// TwinCAT 3 PLC project CNCControl
// ProgramVersion: 3.1.4022.4
// libraries:
//   Tc2_EthernetIP, * (Beckhoff Automation GmbH)
//   Tc2_IoFunctions, * (Beckhoff Automation GmbH)
//   Tc2_Math, * (Beckhoff Automation GmbH)
//   Tc2_Standard, * (Beckhoff Automation GmbH)
//   Tc2_System, * (Beckhoff Automation GmbH)
//   Tc2_Utilities, * (Beckhoff Automation GmbH)
//   Tc3_Module, * (Beckhoff Automation GmbH)
// project tree:
//   DUTs/ E_CIA402State.TcDUT (not stored), E_PIDOptimizationStage.TcDUT (not stored), E_PIDOptimizationType.TcDUT
//   / EveryHundredMilliseconds.TcTTO, EveryMS.TcTTO, MainCNCControl.TcTTO
//   GVLs/ Constants.TcGVL
//   POUs/ MAIN.TcPOU
//   POUs/SpindleSpeed/ AnalogDemandedSpeedCalculator.TcPOU, AnalogPrescaledSpeedCalculator.TcPOU, DemandedSpeedInterface.TcIO, DemandedSpeedTask.TcPOU, PWMDemandedSpeedCalculator.TcPOU, SpindleSpeedCalculator.TcPOU
//   POUs/Spindle/ SpindleCIA402Velocity.TcPOU, SpindleController.TcIO, SpindleDeltaVFDOverEIP.TcPOU
//   POUs/Utilities/ FB_FreqMeasure.TcPOU, FB_MovingAverageUInt.TcPOU, FB_MovingAverageReal.TcPOU, FB_OptimizePID.TcPOU, FB_ScaleBetween.TcPOU
//   POUs/Vacuum/ VacuumATV71Ethercat.TcPOU, FB_GetVacuumAMSID.TcPOU (not stored), ToshibaP9VacuumPressureGetter.TcPOU (not stored), VacuumController.TcIO
// real-time tasks:
//   TASK EveryHundredMilliseconds: cycle T#100000us, priority 10, ADS port 350
//   TASK MainCNCControl: cycle T#1ms, priority 6, ADS port 351
//   TASK EveryMS: cycle T#1ms, priority 4, ADS port 352
// I/O:
//   DEVICE Device 1 (EtherCAT), AmsNetId 192.168.1.51.2.1
//     Box 16 (ATV71 EtherCAT) [ATV71 EtherCAT]
//     HITECO UE-1F 6.6 Spindle [KEB_F6_drive_unit_EtherCAT]
//     Term 1 (EK1100) [EK1100 EtherCAT Coupler (2A E-Bus)]
//       Term 3 (EL1502) [EL1502 2Ch. +/- Counter 24V, 100kHz]
//       Term 4 (EL1809) [EL1809 16Ch. Dig. Input 24V, 3ms]
//       Term 5 (EL1889) [EL1889 16Ch. Dig. Input 24V, 3ms, negative]
//       Term 15 (EL1018) [EL1018 8Ch. Dig. Input 24V, 10µs]
//       Term 20 (EL9110) [EL9110 Power Supplier with LED (24V, Diagnostics)]
//       Term 19 (EL2622) [EL2622 2Ch. Relay Output, NO (230V AC / 30V DC)]
//       Term 26 (EL6070) [EL6070 1Ch. Licensing-Terminal]
//       Term 6 (EL9400) [EL9400 E-Bus Power Supplier]
//       Term 27 (EL1262-0050) [EL1262-0050 2Ch. Dig. Input 5V, 1µs, DC Oversample]
//       Term 7 (EL2124) [EL2124 4Ch. Dig. Output 5V, 20mA]
//       Term 8 (EL2124) [EL2124 4Ch. Dig. Output 5V, 20mA]
//       Term 9 (EL2124) [EL2124 4Ch. Dig. Output 5V, 20mA]
//       Term 10 (EL1124) [EL1124 4Ch. Dig. Input 5V, 10µs, Sensor Power]
//       Term 11 (EL1124) [EL1124 4Ch. Dig. Input 5V, 10µs, Sensor Power]
//       Term 12 (EL9011) [EL9011 End Terminal]
//   DEVICE Device 2 (TC3 EIP Scanner), AmsNetId 192.168.1.51.3.1
//     Box 12 (Nitra CMV EtherNet/IP) // <INFO> </INFO> <EDS> C:\TwinCAT\3.1\Config\Io\EtherNetIP\nitraethernetip.eds </EDS>
//     Box 13 (IPE001Z) (disabled) // <INFO> </INFO> <EDS> C:\TwinCAT\3.1\Config\Io\EtherNetIP\IPE001Z_AS1.eds </EDS>
//     Box 2 (CMM-EIP01) (disabled) // <INFO> </INFO> <EDS> C:\TwinCAT\3.1\Config\Io\EtherNetIP\031F000C010400010001.eds </EDS>
// variable links:
//   CNCControl/CNCControl Instance <-> Device 1 (EtherCAT)/Box 16 (ATV71 EtherCAT)
//     MainCNCControl Inputs/MAIN.VacuumControl.iAnalogInput2ScaledValue <-> Inputs/MAIN.VacuumControl.iAnalogInput2ScaledValue
//     MainCNCControl Inputs/MAIN.VacuumControl.iOutputFrequency <-> Inputs/MAIN.VacuumControl.iOutputFrequency
//     MainCNCControl Inputs/MAIN.VacuumControl.iOutputVelocity <-> Inputs/MAIN.VacuumControl.iOutputVelocity
//     MainCNCControl Inputs/MAIN.VacuumControl.iPIDRegulatorFeedback <-> Inputs/MAIN.VacuumControl.iPIDRegulatorFeedback
//     MainCNCControl Inputs/MAIN.VacuumControl.iPIDRegulatorOutput <-> Inputs/MAIN.VacuumControl.iPIDRegulatorOutput
//     MainCNCControl Inputs/MAIN.VacuumControl.iStatusWord <-> Inputs/MAIN.VacuumControl.iStatusWord
//     MainCNCControl Outputs/MAIN.VacuumControl.oMotorFrequency <-> Outputs/MAIN.VacuumControl.oMotorFrequency
//     MainCNCControl Outputs/MAIN.VacuumControl.oVacuumControl <-> Outputs/MAIN.VacuumControl.oVacuumControl
//     MainCNCControl Outputs/MAIN.VacuumControl.oVacuumPressureRequested <-> Outputs/MAIN.VacuumControl.oVacuumPressureRequested
//   CNCControl/CNCControl Instance <-> Device 1 (EtherCAT)/HITECO UE-1F 6.6 Spindle
//     MainCNCControl Inputs/MAIN.SpindleControl.iStatusWord <-> Inputs/statusword [0x6041.0]
//     MainCNCControl Outputs/MAIN.SpindleControl.oControlWord <-> Outputs/controlword [0x6040.0]
//     MainCNCControl Outputs/MAIN.SpindleControl.oTargetVelocity <-> Outputs/vl target velocity [0x6042.0]
//   CNCControl/CNCControl Instance <-> Device 1 (EtherCAT)/Term 1 (EK1100)/Term 11 (EL1124)
//     MainCNCControl Inputs/MAIN.iPCCoolantOn <-> Channel 4/MAIN.iPCCoolantOn
//     MainCNCControl Inputs/MAIN.iPCSpindleOn <-> Channel 1/MAIN.iPCSpindleOn
//     MainCNCControl Inputs/MAIN.iPCToolRelease <-> Channel 3/MAIN.iPCToolRelease
//     MainCNCControl Inputs/MAIN.iPCVacuumOn <-> Channel 2/MAIN.iPCVacuumOn
//   CNCControl/CNCControl Instance <-> Device 1 (EtherCAT)/Term 1 (EK1100)/Term 15 (EL1018)
//     MainCNCControl Inputs/MAIN.iProbe <-> Channel 1/MAIN.iProbe
//   CNCControl/CNCControl Instance <-> Device 1 (EtherCAT)/Term 1 (EK1100)/Term 19 (EL2622)
//     MainCNCControl Outputs/MAIN.oZAxisBrakeRelay <-> Channel 1/MAIN.oZAxisBrakeRelay
//   CNCControl/CNCControl Instance <-> Device 1 (EtherCAT)/Term 1 (EK1100)/Term 27 (EL1262-0050)
//     EveryMS Inputs/DemandedSpeedTask.DemandedSpeedImpl.iInputSpeedBits[{1..125}] <-> Ch1 Input {0..124}/Ch1 Input  (125 links)
//   CNCControl/CNCControl Instance <-> Device 1 (EtherCAT)/Term 1 (EK1100)/Term 3 (EL1502)
//     EveryHundredMilliseconds Inputs/SpindleSpeedCalculator.CounterValue <-> CNT Inputs Channel 1/Counter value
//   CNCControl/CNCControl Instance <-> Device 1 (EtherCAT)/Term 1 (EK1100)/Term 4 (EL1809)
//     MainCNCControl Inputs/MAIN.iAirPressureSensor <-> Channel 1/MAIN.iPressureSensor
//     MainCNCControl Inputs/MAIN.iS1ToolPresence <-> Channel 5/MAIN.iS1ToolPresence
//     MainCNCControl Inputs/MAIN.iS2ColletOpen <-> Channel 4/MAIN.iS2ColletOpen
//     MainCNCControl Inputs/MAIN.iSpindleOverTemp <-> Channel 3/MAIN.iSpindleOverTemp
//     MainCNCControl Inputs/MAIN.iSpindleToolReleaseButton <-> Channel 2/MAIN.iSpindleToolReleaseButton
//   CNCControl/CNCControl Instance <-> Device 1 (EtherCAT)/Term 1 (EK1100)/Term 5 (EL1889)
//     MainCNCControl Inputs/MAIN.iAAxisAlarm <-> Channel 5/Input
//     MainCNCControl Inputs/MAIN.iXAxisAlarm <-> Channel 2/MAIN.iXAxisAlarm
//     MainCNCControl Inputs/MAIN.iYAxisAlarm <-> Channel 1/MAIN.iYAxisAlarm
//     MainCNCControl Inputs/MAIN.iZAxisAlarm <-> Channel 3/MAIN.iZAxisAlarm
//     MainCNCControl Inputs/MAIN.iZAxisBrakeOff <-> Channel 4/MAIN.iZAxisBrakeOff
//   CNCControl/CNCControl Instance <-> Device 1 (EtherCAT)/Term 1 (EK1100)/Term 7 (EL2124)
//     MainCNCControl Outputs/MAIN.oPCToolPresence <-> Channel 4/MAIN.PCToolPresence
//   CNCControl/CNCControl Instance <-> Device 1 (EtherCAT)/Term 1 (EK1100)/Term 8 (EL2124)
//     MainCNCControl Outputs/MAIN.oPCColletOpen <-> Channel 2/MAIN.oPCColletOpen
//     MainCNCControl Outputs/MAIN.oPCServoAlarm <-> Channel 1/MAIN.oPCServoAlarm
//     MainCNCControl Outputs/MAIN.oPCSpindleStopped <-> Channel 3/MAIN.oPCSpindleStopped
//     MainCNCControl Outputs/MAIN.oPCVacuumPressureGood <-> Channel 4/MAIN.oPCVacuumPressureGood
//   CNCControl/CNCControl Instance <-> Device 1 (EtherCAT)/Term 1 (EK1100)/Term 9 (EL2124)
//     MainCNCControl Outputs/MAIN.oPCAirPressure <-> Channel 1/MAIN.oPCAirPressure
//     MainCNCControl Outputs/MAIN.oPCProbe <-> Channel 2/MAIN.oPCProbe
//     MainCNCControl Outputs/MAIN.oPCSpindleOverTemp <-> Channel 4/MAIN.oPCSpindleOverTemp
//     MainCNCControl Outputs/MAIN.oPCSpindleSpeedOK <-> Channel 3/MAIN.oPCSpindleSpeedOK
//   CNCControl/CNCControl Instance <-> Device 2 (TC3 EIP Scanner)/Box 12 (Nitra CMV EtherNet/IP)
//     MainCNCControl Outputs/MAIN.oValveControl <-> Connection 1 (Input/Output)/Outputs/MAIN.oValveControl

CONFIGURATION CNCControl
    RESOURCE PLC ON TwinCAT3
        TASK EveryHundredMilliseconds(INTERVAL := T#100000us, PRIORITY := 10);
        TASK EveryMS(INTERVAL := T#1ms, PRIORITY := 4);
        TASK MainCNCControl(INTERVAL := T#1ms, PRIORITY := 6);
        PROGRAM VacuumPressureGetter WITH EveryHundredMilliseconds : VacuumPressureGetter;
        PROGRAM SpindleSpeedCalculator WITH EveryHundredMilliseconds : SpindleSpeedCalculator;
        PROGRAM DemandedSpeedTask WITH EveryMS : DemandedSpeedTask;
        PROGRAM MAIN WITH MainCNCControl : MAIN;
    END_RESOURCE
END_CONFIGURATION

// ---- DUTs/E_PIDOptimizationType.TcDUT
{attribute 'qualified_only'}
{attribute 'strict'}
TYPE E_PIDOptimizationType :
(
	NoOvershoot,
	SomeOvershoot,
	FastRamp
);
END_TYPE

// ---- GVLs/Constants.TcGVL
{attribute 'qualified_only'}
VAR_GLOBAL CONSTANT
	// Number of RPM per HZ in the VFD
	RPMPerHZ : UINT := 30;
	// VFD frequency precision in 1/X of 1 HZ. So 10 means it can do 1/10th of a HZ
	VFDHZPrecision : UINT := 10;
	// Minimum VFD RPM increment based on RPM per HZ and precision
	VFDMinRPMIncrement : UINT := TO_UINT(RPMPerHZ / VFDHZPrecision);
	// One second in microseconds
	OneSecondInUs : UDINT := 1000000;
END_VAR

// ---- POUs/SpindleSpeed/DemandedSpeedInterface.TcIO
INTERFACE DemandedSpeedInterface

METHOD GetSpeed : UINT
END_METHOD

END_INTERFACE

// ---- POUs/Spindle/SpindleController.TcIO
INTERFACE SpindleController

METHOD Run : BOOL
END_METHOD

METHOD SetDirection : BOOL
VAR_INPUT
	// Set the spindle rotation direction
	Reverse : BOOL;
END_VAR
END_METHOD

METHOD SetSpeed : BOOL
VAR_INPUT
	Speed : UINT;
END_VAR
END_METHOD

METHOD Stop : BOOL
END_METHOD

END_INTERFACE

// ---- POUs/Vacuum/VacuumController.TcIO
INTERFACE VacuumController

METHOD GetCurrentPressure : REAL
END_METHOD

METHOD Run : BOOL
END_METHOD

METHOD SetPressureRequired : BOOL
VAR_INPUT
	Pressure : REAL;
END_VAR
END_METHOD

METHOD Stop : BOOL
END_METHOD

END_INTERFACE

// ---- POUs/SpindleSpeed/SpindleSpeedCalculator.TcPOU
PROGRAM SpindleSpeedCalculator
VAR
	// Spindle speed in RPM
	{attribute 'UserUnit' := '<AngularVelocity, RPM, RPM, 9.549296596425, 0, 0 >'}
	SpindleSpeed : LREAL;
	// Current pulse count value from the counter
	PulseCount: UINT;
	// Counter value from previous time we read the counter
	LastCounterValue: UDINT;
	// Counter value from counter
	CounterValue AT %I*: UDINT;
	// Array of spindle speeds
	SpindleSpeeds : ARRAY[0..4] OF LREAL;
	MovingAverage : FB_MovingAverageReal;
END_VAR
VAR_TEMP
	TempSpindleSpeed: REAL;
END_VAR
VAR CONSTANT
	// Pulses per revolution of the spindle sensor
	PulsesPerRevolution : UINT := 2;
	// Task cycles per minute - task runs every 100ms
	TaskCyclesPerMinute : UINT := 600;
END_VAR

// Convert counter value to pulses since last cycle
PulseCount := TO_UINT(CounterValue - LastCounterValue);
LastCounterValue := CounterValue;
// Extrapolate how pulses many would have occurred in a minute, then divide by pulses per revolution to get RPM.
TempSpindleSpeed := (TO_REAL(PulseCount) * TaskCyclesPerMinute) / PulsesPerRevolution;
MovingAverage(ValueToAdd := TempSpindleSpeed,
			  AverageArray := SpindleSpeeds);
SpindleSpeed := MovingAverage.CurrentValue;

END_PROGRAM

// ---- POUs/Utilities/FB_MovingAverageReal.TcPOU
FUNCTION_BLOCK FB_MovingAverageReal
VAR_INPUT
	ValueToAdd : LREAL;
END_VAR
VAR_IN_OUT
	AverageArray  : ARRAY [*] OF LREAL;
END_VAR
VAR_OUTPUT
	CurrentValue : LREAL;
END_VAR
VAR
	CurrentIndex : UINT;
	NumValues: UINT;
END_VAR
VAR_TEMP
	Counted : UINT;
	I: DINT;
	Sum: LREAL;
	ArrayLength : UINT;
END_VAR

// Compute average over array.
// The order of this addition and MOD are important to avoid going out of bounds.
// NOTE: We deliberately do not try to account for underfilling the array.
ArrayLength := TO_UINT(UPPER_BOUND(AverageArray, 1) - LOWER_BOUND(AverageArray, 1) + 1);
AverageArray[CurrentIndex] := ValueToAdd;
CurrentIndex := CurrentIndex + 1;
CurrentIndex := CurrentIndex MOD ArrayLength;
NumValues := MIN(NumValues + 1 , ArrayLength);
IF NumValues > 0 THEN
	FOR I := LOWER_BOUND(AverageArray, 1) TO UPPER_BOUND(AverageArray, 1) BY 1 DO
		Sum := Sum + AverageArray[I];
		Counted := Counted + 1;
		// Don't count more than the number of values
		IF Counted > NumValues THEN
			EXIT;
		END_IF
	END_FOR
END_IF
CurrentValue := TO_REAL(Sum / NumValues);

END_FUNCTION_BLOCK

// ---- POUs/SpindleSpeed/DemandedSpeedTask.TcPOU
PROGRAM DemandedSpeedTask
VAR
	{attribute 'UserUnit' := '<AngularVelocity, RPM, RPM, 9.549296596425, 0, 0 >'}
	DemandedSpeed : UINT;
	DemandedSpeedImpl : PWMDemandedSpeedCalculator;
END_VAR

DemandedSpeed := DemandedSpeedImpl.GetSpeed();

END_PROGRAM

// ---- POUs/SpindleSpeed/PWMDemandedSpeedCalculator.TcPOU
FUNCTION_BLOCK FINAL PWMDemandedSpeedCalculator IMPLEMENTS DemandedSpeedInterface
VAR
	iInputSpeedBits AT %I* : ARRAY [1..BitArraySize] OF BYTE;
END_VAR
VAR CONSTANT
	// Array Length
	BitArraySize : UINT := 125;
	// PWM frequency
	PWMFrequency : UINT := 200;
    // PWM period
	PWMPeriod : REAL := 1 / PWMFrequency;
	// Microseconds in Frequency
	UsInFrequency : UDINT :=  Constants.OneSecondInUs / PWMFrequency;	
END_VAR

METHOD GetSpeed : UINT
VAR_INST
	TempSpindleSpeed : UINT;
	LastDemandedSpeed : UINT;
	TotalOnTime : UDINT;
	TotalOffTime : UDINT;
	DutyCycle : LREAL;
	DutyCycles : ARRAY [0..20] OF LREAL;
	MovingAverage : FB_MovingAverageReal;
	Scaling : FB_ScaleBetween;
END_VAR
VAR
	I : UINT;	
	J: UINT;
	BitMask : UINT;
	MaskedBit : BOOL;
END_VAR
// The input here is a PWM signal with a frequency of 200, a low of 1% duty, and a high of 95% duty.
// Basic Calculation for PWM pulses

 FOR I := 1 TO BitArraySize BY 1 DO
	 FOR J := 0 TO 7 BY 1 DO
		BitMask := SHL(1, J);
		MaskedBit := TO_BOOL(iInputSpeedBits[I] AND BitMask);
		IF MaskedBit THEN
			TotalOnTime := TotalOnTime + 1;
		ELSE
			TotalOffTime := TotalOffTime + 1; 
		END_IF
		// Stop at the end of the period
		IF (TotalOnTime + TotalOffTime) > UsInFrequency THEN
			EXIT;
		END_IF 
	 END_FOR
 END_FOR
 
// See if the period is up
IF (TotalOnTime + TotalOffTime) > UsInFrequency  THEN
	DutyCycle := TO_LREAL(TotalOnTime) / TO_LREAL(TotalOnTime + TotalOffTime);
	TotalOnTime := 0;
	TotalOffTime := 0;
	// Average the duty cycle and then scale the average
	MovingAverage(ValueToAdd := DutyCycle, 
				  AverageArray := DutyCycles);
	Scaling(RawValue:=MovingAverage.CurrentValue, RawValueMin:=0.0, 
					  RawValueMax:=1, ScaledValueMin:=0,
					  ScaledValueMax:=24000);
	LastDemandedSpeed := TO_UINT(Scaling.ScaledValue);
	// Make sure demanded speed is some increment of what the VFD can do. 
	LastDemandedSpeed := (LastDemandedSpeed / Constants.VFDMinRPMIncrement) * Constants.VFDMinRPMIncrement;
END_IF
GetSpeed := LastDemandedSpeed;
END_METHOD

END_FUNCTION_BLOCK

// ---- POUs/Utilities/FB_ScaleBetween.TcPOU
FUNCTION_BLOCK FB_ScaleBetween
VAR_INPUT
	RawValue : LREAL;
	RawValueMin: LREAL;
	RawValueMax : LREAL;
	ScaledValueMin : LREAL;
	ScaledValueMax : LREAL;
END_VAR
VAR_OUTPUT
	ScaledValue : LREAL;
END_VAR
VAR
END_VAR

ScaledValue :=  (((ScaledValueMax-ScaledValueMin) * (RawValue - RawValueMin)) / (RawValueMax - RawValueMin)) + ScaledValueMin;
ScaledValue := LIMIT(ScaledValueMin, ScaledValue, ScaledValueMax);

END_FUNCTION_BLOCK

// ---- POUs/MAIN.TcPOU
PROGRAM MAIN
VAR
	{region "Servo handling variables"}
	// Alarm inputs from Servos
  	iXAxisAlarm AT %I*:BOOL;
  	iYAxisAlarm AT %I*:BOOL;
  	iZAxisAlarm AT %I*:BOOL;
  	iAAxisAlarm AT %I*:BOOL;
  	// Alarm Output to PC pin 8
  	oPCServoAlarm AT %Q*:BOOL;
  	// Whether servo thinks Z Axis break should be off
  	iZAxisBrakeOff AT %I*:BOOL;
	// Relay output controlling Z Axis Brake
	oZAxisBrakeRelay AT %Q*: BOOL;
    {endregion}
	{region "Probe, Air Pressure, Coolant"}
	// Digital Probe Trigger output to PC pin 29
	oPCProbe AT %Q*: BOOL;
	// Digital Probe Input (Normally Closed)
	iProbe AT %I*: BOOL := TRUE;
	// Air Pressure >90psi signal to PC pin 10
	oPCAirPressure AT %Q*: BOOL;
	// Air Pressure >90psi signal from sensor.  The sensor triggers as pressure is rising past 90psi
	iAirPressureSensor AT %I*: BOOL;
	// Control of NITRA Valves over ethernet/ip	 
	oValveControl AT %Q* : NitraValves; 
	// Turn on coolant signal from PC
	iPCCoolantOn AT %I* : BOOL;
	{endregion}
	{region "Vacuum"}
	VacuumControl: VacuumATV71Ethercat;
	 // Turn on vacuum signal from PC
	iPCVacuumOn AT %I* : BOOL;
	// Vacuum Pressure good output to PC Pin 7
	oPCVacuumPressureGood AT %Q*: BOOL;
	{endregion}
	{endregion}
	{endregion}
	{region "Spindle variables"}
	{region "Spindle Speed Handling"}
	// True if spindle is at less than 1 RPM
	SpindleStopped : BOOL;
	// Spindle stopped output to PC pin 1
	oPCSpindleStopped AT %Q* : BOOL;
	// Spindle within 5% of speed to PC Pin 28
	oPCSpindleSpeedOK AT %Q* : BOOL;
	{endregion}
	{region "Spindle Tool Change handling"}
	// Tool Release Button on Spindle
	iSpindleToolReleaseButton AT %I*: BOOL;
	// Tool Release from PC Pin 24
	iPCToolRelease AT %I*: BOOL;
	// Tool Presence to PC Pin 2
	oPCToolPresence AT %Q* : BOOL;
	// S1 Tool Presence sensor from the spindle
	iS1ToolPresence AT %I* : BOOL;
	// Collet Open to PC Pin 9
	oPCColletOpen AT %Q* : BOOL;
	// S2 Collet Open sensor from the spindle
	iS2ColletOpen AT %I* : BOOL;	 
	// Spindle over temperature to PC Pin 27
	oPCSpindleOverTemp AT %Q* : BOOL;
	// Spindle over temperature relay
	iSpindleOverTemp AT %I* : BOOL;
	// Turn spindle on input from PC
	iPCSpindleOn AT %I* : BOOL;
	SpindleControl : SpindleCIA402Velocity;
	{endregion}
	{endregion}
	{region "Input Debouncers"}
	(* The 5V input has a ridiculously fast time - a few nanoseconds.
	   Therefore, we debounce it *)
	CoolantOnDebounced : TON;
	SpindleOnDebounced : TON;
	ToolReleaseDebounced : TON;	
	VacuumOnDebounced : TON;
	{endregion}
END_VAR
VAR CONSTANT
	// Minimum PSI at which vacuum holding is viable for workpiece
	GoodVacuumPressure : REAL := 10.0;
END_VAR

CoolantOnDebounced(IN := iPCCoolantOn, PT := T#3MS);
SpindleOnDebounced(IN := iPCSpindleOn, PT := T#3MS);
ToolReleaseDebounced(IN := iPCToolRelease, PT := T#3MS);
VacuumOnDebounced(IN := iPCVacuumOn, PT := T#3MS);

{region "Servo handling"}
// Servo Alarm
	// The servo alarm inputs are normally closed
	oPCServoAlarm := NOT (iXAxisAlarm AND_THEN iYAxisAlarm AND_THEN iZAxisAlarm AND_THEN iAAxisAlarm);

// Servo Brake	 
	oZAxisBrakeRelay := iZAxisBrakeOff;
{endregion}

{region "Probe, Air Pressure, Coolant, Vacuum"}
// Probe control
	oPCProbe := NOT iProbe;

// Pressure Control
	oPCAirPressure := iAirPressureSensor;

// Coolant control
	oValveControl.Coolant := CoolantOnDebounced.Q;

// Vacuum Control
	IF VacuumOnDebounced.Q THEN
		VacuumControl.Run();
	ELSE 
		VacuumControl.Stop();
	END_IF
	oPCVacuumPressureGood := VacuumControl.GetCurrentPressure() >= GoodVacuumPressure;

{endregion}
{region "Spindle handling"}
// Spindle Speed Handling
	// Spindle is stopped if it is under 1RPM
	SpindleStopped := SpindleSpeedCalculator.SpindleSpeed <= 1.0;
	oPCSpindleStopped := SpindleStopped;
	// Calculate whether spindle is up to speed.  We will only say it is up to speed if it is on.
	oPCSpindleSpeedOK := SpindleOnDebounced.Q AND_THEN (SpindleSpeedCalculator.SpindleSpeed  >= (0.95 * TO_REAL(DemandedSpeedTask.DemandedSpeed)));

// Spindle control handling
	 // NOTE: HSK-F63 spindles may not be spun while the tool is not present
	 IF NOT (SpindleOnDebounced.Q AND iS1ToolPresence) THEN
	 	SpindleControl.SetSpeed(0);
		SpindleControl.Stop();
	 ELSIF SpindleOnDebounced.Q AND iS1ToolPresence THEN	  
	 	SpindleControl.SetSpeed(DemandedSpeedTask.DemandedSpeed);
		SpindleControl.Run();
	 END_IF
		  
// Spindle Tool Change handling
	oPCToolPresence := iS1ToolPresence;
	oPCColletOpen := iS2ColletOpen;
	oPCSpindleOverTemp := iSpindleOverTemp;
	oValveControl.ToolRelease := (iAirPressureSensor AND_THEN SpindleStopped) AND_THEN (ToolReleaseDebounced.Q OR iSpindleToolReleaseButton); 		  

{endregion}		  
{endregion}

END_PROGRAM

// ---- POUs/Vacuum/VacuumATV71Ethercat.TcPOU
FUNCTION_BLOCK VacuumATV71Ethercat IMPLEMENTS  VacuumController
VAR_INPUT
END_VAR
VAR_OUTPUT
END_VAR
VAR
	// Vacuum Control Output
	oVacuumControl AT %Q* : ST_ATV71CommandWord;	
	// Vacuum Pressure requested from VFD - in tenths of a psi from 0 to 1450
	oVacuumPressureRequested AT %Q* : UINT;
		 
	{region "Input Vacuum Data"}
	iStatusWord AT %I* : UINT;
	{attribute 'BaseUnit' := '<RPM, 1, 0, 0>'}
	iOutputVelocity AT %I* : UINT;
	iAnalogInput2ScaledValue AT %I* : UINT;
	{attribute 'UserUnit' := '<Pressure, PSI, PSI, 6894.7572932, 0, centi>'}
	iPIDRegulatorFeedback AT %I* : UINT;
	iPIDRegulatorOutput AT %I* : UINT;
	{attribute 'BaseUnit' := '<Frequency, 0.1, 0, 0>'}
	iOutputFrequency AT %I* : UINT;
	{endregion}
	oMotorFrequency AT %Q* : UINT;
	//	PidOptimizer : FB_OptimizePID;
END_VAR

METHOD GetCurrentPressure : REAL
GetCurrentPressure := TO_REAL(iPIDRegulatorFeedback) / 100;
END_METHOD

METHOD Run : BOOL
oVacuumControl.Forward := TRUE;
oVacuumControl.Reverse := FALSE;
oVacuumControl.PidIntegralOff := FALSE;
	
	(* PID optimization
	IF VacuumOnDebounced.Q THEN
		IF NOT PidOptimizer.TuningDone THEN
			PidOptimizer(Enable := TRUE,
						 ProcessSetpoint := 2500,
						 ProcessValue := iAnalogInput2ScaledValue,
						 NumCycles := 10,
						 Reset := FALSE,
						 ControlLowVal := 5,
						 ControlHighVal := 60,
						 PIDType := E_PIDOptimizationType.FastRamp);
			oMotorFrequency := TO_UINT(PidOptimizer.ControlValue*10);
			IF PidOptimizer.TuningDone THEN
				ADSLOGLREAL(TC2_Utilities.ADSLOG_MSGTYPE_LOG, 'Kp value is %f', PidOptimizer.Kp);
				ADSLOGLREAL(TC2_Utilities.ADSLOG_MSGTYPE_LOG, 'Ki value is %f', PidOptimizer.Ki);
				ADSLOGLREAL(TC2_Utilities.ADSLOG_MSGTYPE_LOG, 'Kd value is %f', PidOptimizer.Kd);
				ADSLOGLREAL(TC2_Utilities.ADSLOG_MSGTYPE_LOG, 'Ku value is %f', PidOptimizer.Ku);
				ADSLOGLREAL(TC2_Utilities.ADSLOG_MSGTYPE_LOG, 'Tu value is %f', PidOptimizer.Tu);
			END_IF
		END_IF
	END_IF
	*)
END_METHOD

METHOD SetPressureRequired : BOOL
VAR_INPUT
	Pressure	: REAL;
END_VAR
oVacuumPressureRequested := TO_UINT(Pressure * 100);
END_METHOD

METHOD Stop : BOOL
oVacuumControl.Forward := TRUE;
oVacuumControl.Reverse := FALSE;
oVacuumControl.PidIntegralOff := FALSE;
END_METHOD

END_FUNCTION_BLOCK

// ---- POUs/Spindle/SpindleCIA402Velocity.TcPOU
FUNCTION_BLOCK FINAL SpindleCIA402Velocity IMPLEMENTS SpindleController

VAR
	oControlWord AT %Q*: ST_CIA402ControlWord;
	iStatusWord AT %I*: UINT;
	oTargetVelocity AT %Q* : INT;
	// Forward/backward is specified by positive or negative speed
	VelocityMultiplier : INT := 1;
END_VAR

METHOD GetState : E_CIA402State
VAR CONSTANT
	NotReadyToSwitchOnValue : UINT := 2#0000_0000_0000_0000;
	NotReadyToSwitchOnMask : UINT := 2#0000_0000_0100_1111;
	SwitchOnDisabledValue : UINT := 2#0000_0000_0100_0000;
	SwitchOnDisabledMask : UINT := NotReadyToSwitchOnMask;
	ReadyToSwitchOnValue : UINT := 2#0000_0000_0010_0001;
	ReadyToSwitchOnMask : UINT := 2#0000_0000_0110_1111;
	SwitchedOnValue : UINT := 2#0000_0000_0010_0011;
	SwitchedOnMask : UINT := ReadyToSwitchOnMask;
	OperationEnabledValue : UINT := 2#0000_0000_0010_0111;
	OperationEnabledMask : UINT := ReadyToSwitchOnMask;
	QuickStopActiveValue : UINT := 2#0000_0000_0000_0111;
	QuickStopActiveMask : UINT := ReadyToSwitchOnMask;
	FaultReactionActiveValue : UINT := 2#0000_0000_0000_1111;
	FaultReactionActiveMask : UINT := 2#0000_0000_0100_1111;
	FaultValue : UINT := 2#0000_0000_0000_1000;
	FaultMask : UINT := FaultReactionActiveMask;
END_VAR
IF (iStatusWord AND NotReadyToSwitchOnMask) = NotReadyToSwitchOnValue THEN
	GetState := E_CIA402State.NotReadyToSwitchOn;
ELSIF (iStatusWord AND SwitchOnDisabledMask) = SwitchOnDisabledValue THEN
	GetState := E_CIA402State.SwitchOnDisabled;
ELSIF (iStatusWord AND ReadyToSwitchOnMask) = ReadyToSwitchOnValue THEN
	GetState := E_CIA402State.ReadyToSwitchOn;
ELSIF (iStatusWord AND SwitchedOnMask) = SwitchedOnValue THEN
	GetState := E_CIA402State.SwitchedOn;
ELSIF (iStatusWord AND OperationEnabledMask) = OperationEnabledValue THEN
	GetState := E_CIA402State.OperationEnabled;
ELSIF (iStatusWord AND QuickStopActiveMask) = QuickStopActiveValue THEN
	GetState := E_CIA402State.QuickStopActive;
ELSIF (iStatusWord AND FaultReactionActiveMask) = FaultReactionActiveValue THEN
	GetState := E_CIA402State.FaultReactionActive;
ELSIF (iStatusWord AND FaultMask) = FaultValue THEN
	GetState := E_CIA402State.Fault;
ELSE
	GetState := E_CIA402State.Unknown_State;
END_IF
END_METHOD

METHOD GetStatus : ST_CIA402StatusWord
VAR_INPUT
END_VAR
MEMCPY(ADR(GetStatus), ADR(iStatusWord), SIZEOF(iStatusWord));
END_METHOD

METHOD Run : BOOL
CASE GetState() OF
	E_CIA402State.SwitchOnDisabled:
		oControlWord.EnableVoltage := TRUE;
	E_CIA402State.ReadyToSwitchOn:
		oControlWord.SwitchOn := TRUE;
	E_CIA402State.SwitchedOn:
		oControlWord.EnableOperation := TRUE;
END_CASE
END_METHOD

METHOD SetDirection : BOOL
VAR_INPUT
	(* Set the spindle rotation direction*)
	Reverse	: BOOL;
END_VAR
IF Reverse THEN
	VelocityMultiplier := -1;
ELSE
	VelocityMultiplier := 1;
END_IF
END_METHOD

METHOD SetSpeed : BOOL
VAR_INPUT
	Speed	: UINT;
END_VAR
oTargetVelocity := TO_INT(LIMIT(0, Speed, 32767)) * VelocityMultiplier;
END_METHOD

METHOD Stop : BOOL
CASE GetState() OF
	E_CIA402State.ReadyToSwitchOn:
		oControlWord.EnableVoltage := FALSE;
	E_CIA402State.SwitchedOn:
		oControlWord.SwitchOn := FALSE;
	E_CIA402State.OperationEnabled :
		oControlWord.EnableOperation := FALSE;
END_CASE
END_METHOD

END_FUNCTION_BLOCK

// ---- POUs/SpindleSpeed/AnalogDemandedSpeedCalculator.TcPOU
FUNCTION_BLOCK FINAL AnalogDemandedSpeedCalculator IMPLEMENTS DemandedSpeedInterface
VAR_INPUT
	// Analog speed as 0-10v from PC Pin 13
	iAnalogSpeedVoltage AT %I*: UINT;
END_VAR

METHOD GetSpeed : UINT
VAR_INST
	// Array of spindle speeds
	SpindleSpeeds : ARRAY[0..10] OF UINT;
	MovingAverage : FB_MovingAverageUInt;
	Scaling : FB_ScaleBetween;
END_VAR
Scaling(RawValue:=iAnalogSpeedVoltage, RawValueMin:=5, 
							RawValueMax:=31900, ScaledValueMin:=0,
							ScaledValueMax:=24000);
// Round value to nearest 60
GetSpeed := TO_UINT(Scaling.ScaledValue / 60);
GetSpeed := GetSpeed * 60;
MovingAverage(ValueToAdd := GetSpeed,
			  AverageArray := SpindleSpeeds);
GetSpeed := MovingAverage.CurrentValue / 60;
GetSpeed := GetSpeed * 60;
END_METHOD

END_FUNCTION_BLOCK

// ---- POUs/Utilities/FB_MovingAverageUInt.TcPOU

FUNCTION_BLOCK FB_MovingAverageUInt
VAR_INPUT
	// Value to add to the moving average.
	ValueToAdd : UINT;
	// The number of values to store in the array.
	NumValuesToUse : UINT := TO_UINT(UPPER_BOUND(AverageArray, 1) - LOWER_BOUND(AverageArray, 1) + 1);
END_VAR
VAR_IN_OUT
	AverageArray  : ARRAY [*] OF UINT;
END_VAR
VAR_OUTPUT
	CurrentValue : UINT;
END_VAR
VAR
	CurrentIndex : UINT;
	NumValuesAdded : UINT;
END_VAR
VAR_TEMP
	I: DINT;
	Sum: UDINT;
	ArrayLength : UINT := TO_UINT(UPPER_BOUND(AverageArray, 1) - LOWER_BOUND(AverageArray, 1) + 1);
	Counted: UINT;
END_VAR

// Compute average over array.
// The order of this addition and MOD are important to avoid going out of bounds.
NumValuesToUse := MIN(ArrayLength, NumValuesToUse);
AverageArray[CurrentIndex] := ValueToAdd;
CurrentIndex := CurrentIndex + 1;
CurrentIndex := CurrentIndex MOD NumValuesToUse;
NumValuesAdded := MIN(NumValuesAdded + 1 , NumValuesToUse);
IF NumValuesAdded > 0 THEN
	FOR I := LOWER_BOUND(AverageArray, 1) TO UPPER_BOUND(AverageArray, 1) BY 1 DO
		Sum := Sum + AverageArray[I];
		// Don't count more than the number of values
		IF Counted > NumValuesAdded THEN
			EXIT;
		END_IF
	END_FOR
END_IF
CurrentValue := TO_UINT(Sum / NumValuesAdded);

END_FUNCTION_BLOCK

// ---- POUs/SpindleSpeed/AnalogPrescaledSpeedCalculator.TcPOU
// This version uses the EL3161 and it's built in IIR filter
FUNCTION_BLOCK FINAL AnalogPrescaledSpeedCalculator IMPLEMENTS DemandedSpeedInterface; 
VAR_INPUT
	// Analog speed as 0-10v from PC Pin 13
	iAnalogSpeed AT %I*: INT;
END_VAR

METHOD GetSpeed : UINT
GetSpeed := TO_UINT(LIMIT(0, iAnalogSpeed, 24000))
END_METHOD

END_FUNCTION_BLOCK

// ---- POUs/Spindle/SpindleDeltaVFDOverEIP.TcPOU
FUNCTION_BLOCK FINAL SpindleDeltaVFDOverEIP IMPLEMENTS SpindleControl
VAR
	// Delta VFD control for the spindle
	oSpindleControl AT %Q* : ST_DeltaVFDCommandWord;
	oSpindleFrequency AT %Q* : UINT;
END_VAR
VAR CONSTANT
	// Number of RPM per HZ in the VFD
	RPMPerHZ : UINT := 30;
	// VFD frequency precision in 1/X of 1 HZ. So 10 means it can do 1/10th of a HZ
	VFDHZPrecision : UINT := 10;
	// Minimum VFD RPM increment based on RPM per HZ and precision
	VFDMinRPMIncrement : UINT := TO_UINT(RPMPerHZ / VFDHZPrecision);
END_VAR

METHOD Run : BOOL
oSpindleControl.Stop := FALSE;
oSpindleControl.Run := TRUE;
END_METHOD

METHOD SetDirection : BOOL
VAR_INPUT
	// Set the spindle rotation direction
	Reverse	: BOOL;
END_VAR
IF Reverse THEN
	oSpindleControl.Reverse := TRUE;
	oSpindleControl.Forward := FALSE;
ELSE
	oSpindleControl.Reverse := FALSE;
	oSpindleControl.Forward := TRUE;
END_IF
END_METHOD

METHOD SetSpeed : BOOL
VAR_INPUT
	Speed: UINT;
END_VAR
// The spindle frequency is in increments of 0.1hz
oSpindleFrequency := (SPEED * Constants.VFDHZPrecision) / Constants.RPMPerHZ;
END_METHOD

METHOD Stop : BOOL
oSpindleControl.Stop := TRUE;
oSpindleControl.Run := FALSE;
END_METHOD

END_FUNCTION_BLOCK

// ---- POUs/Utilities/FB_FreqMeasure.TcPOU
FUNCTION_BLOCK FB_FreqMeasure
// This function is the equivalent of FREQ_MEASURE from codesys's utility library
VAR_INPUT
	// Input signal
    IN: BOOL;
	// Number of periods to average the frequency over.
	// Must be between 1 and 100
    PERIODS: INT :=1;
	// Reset all parameters to 0
    RESET: BOOL;
END_VAR
VAR_OUTPUT
	// Frequency in HZ
    OUT: REAL;
	// FALSE until we've measured at least PERIODS periods, or if distance between two rising edges is > 3 * OUT
    VALID: BOOL;
END_VAR
VAR
	RisingEnableEdge: R_TRIG;
	FallingEnableEdge : F_TRIG;
    STARTED: BOOL;
    RISETIME: TIME;
	// Difference in time between current and last rising edge
    DIFF: DINT;
	// Array of time differences for each period
    TIMEDIFF: ARRAY[0..99] OF DINT;
	// How many periods we have counted so far
    COUNT: INT;
	// Current place in the array of time differences
    IDX: INT;
    I: INT;
	SUM: DINT;
	SYSTIMEMS : TIME;          
END_VAR


IF RESET THEN
    VALID := FALSE;
    COUNT := 0;
    IDX := 0;
    STARTED := FALSE;
    OUT := 0;
    RETURN;
END_IF

RisingEnableEdge(CLK := IN);
FallingEnableEdge(CLK := IN);

// We care only about whether we are the beginning or the end of the signal
IF RisingEnableEdge.Q OR FallingEnableEdge.Q THEN
	SYSTIMEMS := ULINT_TO_TIME(F_GetTaskTime() / TC2_Utilities.SYSTEMTIME_TICKSPERMSEC64);
    IF FallingEnableEdge.Q AND STARTED THEN
		DIFF := TIME_TO_DINT(SYSTIMEMS - RISETIME);
		// We assume time never goes backwards for real. Unfortunately, the API of this call does
		// not give us a way to express errors easily.
        IF Diff > 0 THEN
			// Emulate the weird behavior of CODESYS FREQ_MEASURE
			IF VALID AND Diff > 3000 * REAL_TO_DINT(OUT) THEN
				VALID := FALSE;
				COUNT := 0;
				IDX := 0;
				RETURN;
			END_IF
            TIMEDIFF[IDX] := DIFF;
            IDX := (IDX + 1) MOD PERIODS;
            COUNT := MIN(COUNT + 1, PERIODS);
			// Go valid once we have the minimum number of periods to average over.
            IF COUNT = PERIODS THEN
                SUM := 0;
				// Sum first, then convert to real, to minimize error.
                FOR I :=0 TO PERIODS-1 DO
                    SUM := SUM + TIMEDIFF[I];
                END_FOR
                OUT := 1000.0 * PERIODS / DINT_TO_REAL(SUM);
                VALID := TRUE;
            ELSE 
                VALID := FALSE;
            END_IF
        END_IF
		STARTED := FALSE;
		RETURN;
    END_IF
    STARTED := TRUE;
    RISETIME := SYSTIMEMS;
END_IF

END_FUNCTION_BLOCK

// ---- POUs/Utilities/FB_OptimizePID.TcPOU
FUNCTION_BLOCK FB_OptimizePID

VAR_INPUT
	// Starts the sequence on the rising edge
	Enable : BOOL; 
	// Set point 
	ProcessSetpoint : REAL; 
	// Process measurement 
	ProcessValue : REAL;
	// Number of automatic adjustment cycles (minimum 2) 
	NumCycles : INT := 2; 
	// Reset
	Reset : BOOL;
	// Low value for the square wave output
	ControlLowVal : REAL;
	// High value for the square wave output
	ControlHighVal: REAL;
	// PID constants to use
	PIDType: E_PIDOptimizationType;
END_VAR
VAR_OUTPUT
	// End sequence
	TuningDone: BOOL;
	// Square wave output for the exitation of the process
	ControlValue: REAL; 
	// Proportional gain
	Kp: REAL;
	// Integral time in S
	Ki: REAL;
	// Derivative time in s
	Kd: REAL;
	// Ultimate Gain 
	Ku: REAL;
	// Ultimate Period
	Tu: REAL;
END_VAR
VAR
	// Enable trigger
	rTrigEnable : R_TRIG;
	// Amplitude of process variable
	b: REAL;
	// Amplitude of control variable
	a: REAL;
    TuFreq: FB_FreqMeasure;      
    b_Min: REAL;
    b_Max: REAL;
	EndTrigger : R_TRIG;    
    TuningSequence: E_PIDOptimizationStage;
    CycleNumber: INT;
END_VAR
VAR CONSTANT
    PI : REAL := REAL#3.14159265358979323846264338327950288;
	REAL_MAX : REAL :=  3.402823E+38;
	REAL_MIN : REAL :=-3.402823E+38;
END_VAR


IF Reset THEN
    TuningSequence := E_PIDOptimizationStage.Init;
	TuningDone := FALSE;
END_IF;
IF TuningDone THEN
	RETURN;
END_IF

CASE TuningSequence OF
	// Startup - initialize and set to ramp up to setpoint
	E_PIDOptimizationStage.Init: 
		ControlValue := ControlLowVal;
		IF rTrigEnable.Q THEN
			TuFreq(
				IN := FALSE,
				PERIODS := NumCycles,
				RESET := TRUE); 
			b_Min := REAL_MAX ;
			b_Max := REAL_MIN ;
			KP := 0;
			Ki := 0;
			Kd := 0;
			CycleNumber := 0;
			TuningSequence := E_PIDOptimizationStage.RampingUp;
		END_IF;

	// Ramp to setpoint
	E_PIDOptimizationStage.RampingUp:
		ControlValue := ControlHighVal;
		// If we hit the setpoint, transition to ramping down
		IF ProcessValue > ProcessSetpoint THEN
			ControlValue := ControlLowVal;
			CycleNumber := CycleNumber + 1;
			TuningSequence := E_PIDOptimizationStage.RampingDown;
		END_IF;
		
	// Wait for process value to fall below setpoint
	E_PIDOptimizationStage.RampingDown:
		// Once process value falls, either we are done if we hit the cycle count,
		// or we need to start the next cycle.
		IF ProcessValue < ProcessSetpoint THEN
			IF CycleNumber > NumCycles THEN
				TuningSequence := E_PIDOptimizationStage.Done;
			ELSE
				TuningSequence := E_PIDOptimizationStage.RampingUp;
			END_IF;
		END_IF;

END_CASE;


(*Only Start Measuring Min/Max once we've crossed setpoint once this is to make sure we don't take 0 as value*)
IF CycleNumber  > 0  THEN
	b_Min := MIN(b_Min, ProcessValue);
	b_Max := MAX(b_Max, ProcessValue);
	
	
	TuFreq(
		IN := ProcessValue > ProcessSetpoint,
		PERIODS := NumCycles,
		RESET := FALSE); 
	// We don't check the error becuase i'm lazy. In a real system, if the TuFreq goes invalid, it means the data is screwed up and you need to do something.

END_IF
EndTrigger(CLK := TuningSequence = E_PIDOptimizationStage.Done AND TuFreq.OUT <> 0);
IF EndTrigger.Q THEN
    // Calculate amplitude of control variable
    a := ControlHighVal - ControlLowVal;

	// Calculate amplitude of process variable
    b := b_Max - b_Min;

    // Calculate ultimate period and gain
    Ku := (4 * b)/(PI * a);
    Tu := 1 / TuFreq.OUT;

    CASE PIDType OF
    E_PIDOptimizationType.PessenIntegralRule:
        Kp := 0.7 * Ku;
        Ki := (1.75 * Kp) / Tu;
        Kd := 3* Kp * (Tu/20.0);

    E_PIDOptimizationType.SomeOvershoot:
        Kp := Ku /3.0;
        Ki := (2/3.0) * Ku / Tu ;
        Kd := Ku * Tu  / 10.0;

    E_PIDOptimizationType.NoOvershoot:
        Kp := 0.2 * Ku ;
        Ki := 2 * Ku / Tu  / 5.0;
        Kd := 2* Ku * Tu / 3.0;
    END_CASE;
    
    TuningDone := TRUE;
    TuningSequence := E_PIDOptimizationStage.Init;

END_IF;
rTrigEnable(CLK := Enable);

END_FUNCTION_BLOCK
